INTERFACE I_Payload_B EXTENDS I_Payload

END_INTERFACE

(* stored: Version 1.1.0.1, ProductVersion 3.1.4024.2
   Itf I_Payload_B: Id {eb1c8484-4281-4f0d-b343-29268664d603} *)
